// TwinCAT 3 PLC project protobuf
// Title: protobuf
// Company: TcHaxx
// Author: densogiaichned
// ProjectVersion: 0.0.0.0
// Description: Protocol Buffers for TwinCAT 3
// ProgramVersion: 3.1.4026.20
// libraries:
//   Tc2_Standard, * (Beckhoff Automation GmbH)
//   Tc2_System, * (Beckhoff Automation GmbH)
//   Tc2_Utilities, * (Beckhoff Automation GmbH)
//   TcUnit, * (www.tcunit.org)
// project tree:
//   DUTs/ E_CodedInputStreamErrorCode.TcDUT (not stored), E_CodedOutputStreamErrorCode.TcDUT (not stored), ST_ParseContext.TcDUT (not stored), ST_WriteContext.TcDUT (not stored), ST_Span.TcDUT (not stored), T_ProtobufMaxString.TcDUT (not stored), T_ProtobufRawBuffer.TcDUT (not stored)
//   FieldCodec/ FB_FieldCodec.TcPOU (not stored), FB_FieldCodecFixed32.TcPOU (not stored), FB_FieldCodecFixed64.TcPOU (not stored), FB_FieldCodecDouble.TcPOU (not stored), FB_FieldCodecBool.TcPOU (not stored), FB_FieldCodecEnum.TcPOU, FB_FieldCodecMessage.TcPOU, FB_FieldCodecUInt64.TcPOU (not stored), FB_FieldCodecUInt32.TcPOU (not stored), FB_FieldCodecString.TcPOU (not stored), FB_FieldCodecFloat.TcPOU (not stored), FB_FieldCodecInt32.TcPOU (not stored), FB_FieldCodecSint32.TcPOU (not stored), FB_FieldCodecInt64.TcPOU (not stored), FB_FieldCodecSint64.TcPOU (not stored), FB_FieldCodecBytes.TcPOU (not stored)
//   GVLs/ GCL_PB.TcGVL (not stored), Param_PB.TcGVL (not stored)
//   Helper/DUTs/ ST_VariableLengthArrayInfo.TcDUT (not stored), T_AnyInt.TcDUT (not stored), T_AnyIntOrBit.TcDUT (not stored), T_AnyString.TcDUT (not stored), T_AnyNum.TcDUT (not stored), T_Any.TcDUT (not stored), T_AnyBit.TcDUT (not stored), T_AnyBytes.TcDUT (not stored)
//   Helper/POUs/ F_ParseError.TcPOU (not stored), F_WriteError.TcPOU (not stored), F_ToAnyBit.TcPOU (not stored), F_ToAnyInt.TcPOU (not stored), F_ToAnyBytes.TcPOU (not stored), F_ToAnyType.TcPOU (not stored), F_ToAnyNum.TcPOU (not stored), F_ToAnyString.TcPOU (not stored), F_BufferInfo.TcPOU (not stored), F_WriteToBuffer.TcPOU (not stored), F_ReadFromBuffer.TcPOU (not stored)
//   ITFs/ I_Message.TcIO (not stored), I_FieldCodec.TcIO (not stored), I_RepeatedField.TcIO (not stored), I_ValueReader.TcIO (not stored), I_ValueWriter.TcIO (not stored)
//   ParsingPrimitivesMessages/POUs/ F_ReadMessage.TcPOU, F_ReadRawMessage.TcPOU (not stored), F_SkipLastField.TcPOU (not stored), F_CheckReadEndOfStreamTag.TcPOU (not stored)
//   ParsingPrimitives/DUTs/ E_ParserErrorCode.TcDUT (not stored), ST_ParserInternalState.TcDUT (not stored)
//   ParsingPrimitives/POUs/ F_DecodeZigZag32.TcPOU (not stored), F_DecodeZigZag64.TcPOU (not stored), F_MaybeConsumeTag.TcPOU (not stored), F_ParseDouble.TcPOU (not stored), F_ParseFloat.TcPOU (not stored), F_ParseRawLittleEndian32.TcPOU (not stored), F_ParseLength.TcPOU (not stored), F_ParseRawLittleEndian64.TcPOU (not stored), F_ParseRawVarint64.TcPOU (not stored), F_ParseTag.TcPOU (not stored), F_ParseRawVarint32.TcPOU (not stored), F_PeekTag.TcPOU (not stored), F_ReadBytes.TcPOU (not stored), F_ReadRawByte.TcPOU (not stored), F_ReadRawBytes.TcPOU (not stored), F_ReadStringInternal.TcPOU (not stored), F_SkipRawBytes.TcPOU (not stored), F_ReadRawString.TcPOU (not stored), F_ReadString.TcPOU (not stored)
//   / PlcTask.TcTTO (not stored), PlcTaskUnitTests.TcTTO (not stored)
//   POUs/ComputeSize/ F_ComputeBoolSize.TcPOU (not stored), F_ComputeMessageSize.TcPOU, F_ComputeTagSize.TcPOU (not stored), F_ComputeStringSize.TcPOU (not stored), F_ComputeFixed32Size.TcPOU (not stored), F_ComputeSFixed32Size.TcPOU (not stored), F_ComputeFixed64Size.TcPOU (not stored), F_ComputeSFixed64Size.TcPOU (not stored), F_ComputeInt32Size.TcPOU (not stored), F_ComputeEnumSize.TcPOU, F_ComputeFloatSize.TcPOU (not stored), F_ComputeDoubleSize.TcPOU (not stored), F_ComputeInt64Size.TcPOU (not stored), F_ComputeLengthSize.TcPOU (not stored), F_ComputeBytesSize.TcPOU (not stored), F_ComputeRawVarint64Size.TcPOU (not stored), F_ComputeSInt64Size.TcPOU (not stored), F_ComputeUInt32Size.TcPOU (not stored), F_ComputeRawVarint32Size.TcPOU (not stored), F_ComputeSInt32Size.TcPOU (not stored), F_ComputeUInt64Size.TcPOU (not stored)
//   POUs/ FB_MessageParser.TcPOU (not stored), FB_MessageWriter.TcPOU
//   POUs/ParseContext/ FB_ParseContext.TcPOU
//   POUs/SegmentedBufferHelper/ F_SbhIsReachedLimit.TcPOU (not stored), F_SbhPushLimit.TcPOU (not stored), F_SbhPopLimit.TcPOU (not stored), F_SbhRecomputeBufferSizeAfterLimit.TcPOU (not stored)
//   POUs/Span/ F_SpanFromArray.TcPOU (not stored), F_SpanSlice.TcPOU (not stored)
//   POUs/WriteContext/ FB_WriteContext.TcPOU
//   Project Information/ F_GetCompany.TcPOU (not stored), F_GetTitle.TcPOU (not stored), F_GetVersion.TcPOU (not stored)
//   RepeatedField/ FB_RepeatedField.TcPOU, F_IsPackedRepeatedField.TcPOU (not stored), F_ReadRepeatedField.TcPOU, F_WriteRepeatedField.TcPOU (not stored)
//   WireFormat/DUTs/ E_WireType.TcDUT (not stored)
//   WireFormat/GCLs/ GCL_WireFormat.TcGVL (not stored)
//   WireFormat/POus/ F_GetTagFieldNumber.TcPOU (not stored), F_GetTagWireType.TcPOU (not stored), F_MakeTag.TcPOU (not stored)
//   WritingPrimitivesMessages/POUs/ F_SetMessageValue.TcPOU (not stored), F_WriteMessage.TcPOU, F_WriteRawMessage.TcPOU (not stored)
//   WritingPrimitives/DUTs/ E_WriterErrorCode.TcDUT (not stored), ST_WriterInternalState.TcDUT (not stored)
//   WritingPrimitives/POUs/ F_EncodeZigZag32.TcPOU (not stored), F_EncodeZigZag64.TcPOU (not stored), F_WriteBytes.TcPOU (not stored), F_WriteDouble.TcPOU (not stored), F_WriteFixed32.TcPOU (not stored), F_WriteRawByte.TcPOU (not stored), F_WriteSInt32.TcPOU (not stored), F_WriteSFixed32.TcPOU (not stored), F_WriteFloat.TcPOU (not stored), F_WriteInt32.TcPOU (not stored), F_WriteFixed64.TcPOU (not stored), F_WriteSFixed64.TcPOU (not stored), F_WriteSInt64.TcPOU (not stored), F_WriteRawString.TcPOU (not stored), F_WriteRawTag.TcPOU (not stored), F_WriteUInt32.TcPOU (not stored), F_WriteRawLittleEndian32.TcPOU (not stored), F_WriteLength.TcPOU (not stored), F_WriteRawBytes.TcPOU (not stored), F_WriteRawLittleEndian64.TcPOU (not stored), F_WriteRawVarint32.TcPOU (not stored), F_WriteRawVarint64.TcPOU (not stored), F_WriteString.TcPOU (not stored), F_WriteTag.TcPOU (not stored), F_WriteEnum.TcPOU (not stored), F_WriteUInt64.TcPOU (not stored), F_WriteInt64.TcPOU (not stored)
//   __TESTs/HelperTests/ FB_F_ToAnyBytesTests.TcPOU (not stored), PRG_HelperTests.TcPOU (not stored)
//   __TESTs/EnumTests/ FB_ComputeEnumSizeTests.TcPOU, FB_FieldCodecEnumTests.TcPOU, FB_ReadEnumTests.TcPOU, FB_WriteEnumTests.TcPOU, PRG_EnumTests.TcPOU
//   __TESTs/MessagesTests/DUTs/ ST_Bar.TcDUT (not stored), ST_Baz.TcDUT (not stored), ST_Foo.TcDUT (not stored), ST_Example.TcDUT (not stored)
//   __TESTs/MessagesTests/ FB_MessageTests.TcPOU (not stored), PRG_MessageTests.TcPOU
//   __TESTs/MessagesTests/POUs/ FB_ExampleMessage.TcPOU (not stored), FB_RepeatedStringMessageTests.TcPOU (not stored), FB_RoundTripMessageExampleTest.TcPOU (not stored), FB_ReadMessageErrorTests.TcPOU, FB_TestWrongSizeMessage.TcPOU, FB_WriteMessageSizeTests.TcPOU
//   __TESTs/MessagesTests/POUs/FooBarBaz/ FB_BarMessage.TcPOU (not stored), FB_BazMessage.TcPOU (not stored), FB_FooMessage.TcPOU (not stored)
//   __TESTs/ParsingPrimitivesTests/ FB_DecodeZigZag32Tests.TcPOU (not stored), FB_DecodeZigZag64Tests.TcPOU (not stored), FB_ParseDoubleTests.TcPOU (not stored), FB_ParseFloatTests.TcPOU (not stored), FB_ParseRawVarint32Tests.TcPOU (not stored), FB_ParseRawVarint64Tests.TcPOU (not stored), FB_ReadBytesTests.TcPOU (not stored), FB_ReadRawStringTests.TcPOU (not stored), FB_ReadStringTests.TcPOU (not stored), PRG_ParsingPrimitiveTests.TcPOU (not stored)
//   __TESTs/ PRG_UnitTests.TcPOU
//   Version/ Global_Version.TcGVL (not stored)
//   __TESTs/RepeatedFieldTests/ PRG_RepeatedFieldTests.TcPOU (not stored), FB_TestFixed32Message.TcPOU
//   __TESTs/RepeatedFieldTests/Read/ FB_ReadRepeatedFieldBoolTests.TcPOU (not stored), FB_ReadRepeatedFieldBytesTests.TcPOU (not stored), FB_ReadRepeatedFieldFixed32Tests.TcPOU (not stored), FB_ReadRepeatedFieldFixed64Tests.TcPOU (not stored), FB_ReadRepeatedFieldStringTests.TcPOU (not stored), FB_ReadRepeatedFieldMessageTests.TcPOU, FB_ReadRepeatedFieldUint32Tests.TcPOU (not stored), PRG_ReadRepeatedFieldTests.TcPOU
//   __TESTs/RepeatedFieldTests/RoundTrip/ FB_RoundTripRepeatedFieldUInt32Tests.TcPOU (not stored), FB_RoundTripRepeatedFieldStringTests.TcPOU (not stored), FB_RoundTripRepeatedFieldUInt64Tests.TcPOU (not stored), PRG_RoundTripRepeatedFieldTests.TcPOU (not stored)
//   __TESTs/RepeatedFieldTests/Write/ FB_WriteRepeatedFieldBoolTests.TcPOU (not stored), FB_WriteRepeatedFieldBytesTests.TcPOU (not stored), FB_WriteRepeatedFieldDoubleTests.TcPOU (not stored), FB_WriteRepeatedFieldFixed32Tests.TcPOU (not stored), FB_WriteRepeatedFieldFixed64Tests.TcPOU (not stored), FB_WriteRepeatedFieldFloatTests.TcPOU (not stored), FB_WriteRepeatedFieldInt32Tests.TcPOU (not stored), FB_WriteRepeatedFieldInt64Tests.TcPOU (not stored), FB_WriteRepeatedFieldMessageTests.TcPOU, FB_WriteRepeatedFieldSInt32Tests.TcPOU (not stored), FB_WriteRepeatedFieldSInt64Tests.TcPOU (not stored), FB_WriteRepeatedFieldStringTests.TcPOU (not stored), FB_WriteRepeatedFieldUint32Tests.TcPOU (not stored), FB_WriteRepeatedFieldUint64Tests.TcPOU (not stored), PRG_WriteRepeatedFieldTests.TcPOU (not stored)
//   __TESTs/RoundTripTests/ FB_RoundTripBytesTests.TcPOU (not stored), FB_RoundTripFloatTests.TcPOU (not stored), FB_RoundTripDoubleTests.TcPOU (not stored), FB_RoundTripRawVarint32Tests.TcPOU (not stored), FB_RoundTripRawVarint64Tests.TcPOU (not stored), FB_RoundTripStringTests.TcPOU (not stored), FB_RoundTripTagTests.TcPOU (not stored), FB_RoundTripZigZag32Tests.TcPOU (not stored), FB_RoundTripZigZag64Tests.TcPOU (not stored), PRG_RoundTripTests.TcPOU (not stored)
//   __TESTs/SpanTests/ FB_F_SpanFromArrayTests.TcPOU (not stored), FB_F_SpanSliceTests.TcPOU (not stored), PRG_SpanTests.TcPOU (not stored)
//   __TESTs/WireFormatTests/ FB_MakeTagTests.TcPOU (not stored), PRG_WireFormatTests.TcPOU (not stored)
//   __TESTs/WritingPrimitiveTests/ FB_EncodeZigZag64Tests.TcPOU (not stored), FB_EncodeZigZag32Tests.TcPOU (not stored), FB_WriteBytesTests.TcPOU (not stored), FB_WriteDoubleTests.TcPOU (not stored), FB_WriteRawVarint32Tests.TcPOU (not stored), FB_WriteFloatTests.TcPOU (not stored), FB_WriteRawVarint64Tests.TcPOU (not stored), FB_WriteTagTests.TcPOU (not stored), FB_WriteStringTests.TcPOU (not stored), PRG_WritingPrimitiveTests.TcPOU (not stored)
//   __TESTs/__GENERATED/ E_Color.TcDUT (not stored), E_DataType.TcDUT (not stored), E_Status.TcDUT (not stored), FB_ComplexData.TcPOU (not stored), FB_Device.TcPOU (not stored), FB_Motor.TcPOU (not stored), FB_MotorConfig.TcPOU (not stored), FB_ScalarTypesTest.TcPOU (not stored), FB_SensorReading.TcPOU (not stored), ST_ComplexData.TcDUT (not stored), ST_Device.TcDUT (not stored), ST_Motor.TcDUT (not stored), ST_MotorConfig.TcDUT (not stored), ST_ScalarTypesTest.TcDUT (not stored), ST_SensorReading.TcDUT (not stored)

// ---- FieldCodec/FB_FieldCodecEnum.TcPOU
FUNCTION_BLOCK FB_FieldCodecEnum EXTENDS FB_FieldCodec
VAR_INPUT
END_VAR
VAR_OUTPUT
END_VAR
VAR
    nValue : DINT;
END_VAR

METHOD CalculatePackedDataSize : HRESULT
VAR_INPUT CONSTANT
	anyFirstElem	: T_Any;
	nLength	        : UDINT;
END_VAR
VAR_OUTPUT
    nPackedDataSize : UDINT;
END_VAR
VAR
    anyItem : T_Any;
    i : UDINT;
    nCopySize : UDINT;
    nTmp : DINT;
    retVal : UDINT;
END_VAR
nPackedDataSize := 0;

IF anyFirstElem.pValue = NULL OR anyFirstElem.TypeClass <> __SYSTEM.TYPE_CLASS.TYPE_ENUM THEN
    CalculatePackedDataSize := E_HRESULTAdsErr.INVALIDDATA;
    RETURN;
END_IF

nCopySize := MIN(TO_UDINT(anyFirstElem.diSize), SIZEOF(nTmp));
IF nCopySize = 0 THEN
    CalculatePackedDataSize := E_HRESULTAdsErr.INVALIDDATA;
    RETURN;
END_IF

IF nLength < 1 THEN
    CalculatePackedDataSize := S_OK;
    RETURN;
END_IF

anyItem := anyFirstElem;

FOR i := 0 TO nLength - 1 DO
    anyItem.pValue := anyFirstElem.pValue + (i * TO_UDINT(anyFirstElem.diSize));
    nTmp := 0;
    retVal := MEMCPY(destAddr:= ADR(nTmp), srcAddr:= anyItem.pValue, n:= nCopySize);
    IF retVal = 0 THEN
        CalculatePackedDataSize := E_HRESULTAdsErr.INVALIDDATA;
        RETURN;
    END_IF
    nPackedDataSize := nPackedDataSize + F_ComputeInt32Size(nTmp);
END_FOR

CalculatePackedDataSize := S_OK;
END_METHOD

METHOD IsPackedRepeatedField : BOOL
VAR_INPUT
	nTag	: UDINT;
END_VAR
IsPackedRepeatedField := F_IsPackedRepeatedField(nTag);
END_METHOD


METHOD ValueReader : HRESULT
VAR_IN_OUT
    stCtx : ST_ParseContext;
END_VAR
VAR_OUTPUT
	anyOut	: T_Any;
END_VAR
nValue := 0;
ValueReader := F_ParseRawVarint32(stCtx, nValue);
IF FAILED(ValueReader) THEN
    RETURN;
END_IF

anyOut := F_ToAnyType(anyArg:= nValue);
END_METHOD

METHOD ValueWriter : HRESULT
VAR_IN_OUT
    stCtx  : ST_WriteContext;
END_VAR
VAR_INPUT
	anyIn	: T_ANY;
END_VAR
VAR
    nCopySize : UDINT;
    retVal : UDINT;
END_VAR
IF anyIn.pValue = NULL OR anyIn.TypeClass <> __SYSTEM.TYPE_CLASS.TYPE_ENUM THEN
    ValueWriter := E_HRESULTAdsErr.INVALIDDATA;
    RETURN;
END_IF

nCopySize := MIN(TO_UDINT(anyIn.diSize), SIZEOF(nValue));
IF nCopySize = 0 THEN
    ValueWriter := E_HRESULTAdsErr.INVALIDDATA;
    RETURN;
END_IF

nValue := 0;
retVal := MEMCPY(destAddr:= ADR(nValue), srcAddr:= anyIn.pValue, n:= nCopySize);
IF retVal = 0 THEN
    ValueWriter := E_HRESULTAdsErr.INVALIDDATA;
    RETURN;
END_IF

ValueWriter := F_WriteEnum(stCtx, nValue);
END_METHOD

END_FUNCTION_BLOCK

// ---- FieldCodec/FB_FieldCodecMessage.TcPOU
FUNCTION_BLOCK FB_FieldCodecMessage Extends FB_FieldCodec
VAR_INPUT
END_VAR
VAR_OUTPUT
END_VAR
VAR
END_VAR

{attribute 'analysis' := '-33'}
METHOD CalculatePackedDataSize : HRESULT
VAR_INPUT CONSTANT
	anyFirstElem	: T_Any;
	nLength	        : UDINT;        // items to write
END_VAR
VAR_OUTPUT
    nPackedDataSize : UDINT;
END_VAR
VAR
    anyItem : T_Any;
    i : UDINT;
    eErrorCode : E_WriterErrorCode;
END_VAR
nPackedDataSize := 0;

IF THIS^.ipMessageField = NULL THEN
    CalculatePackedDataSize := E_HRESULTAdsErr.INVALIDDATA;
    RETURN;
END_IF

IF nLength < 1 THEN
    CalculatePackedDataSize := S_OK;
    RETURN;
END_IF

anyItem := anyFirstElem;

FOR i := 0 TO nLength - 1 DO
    anyItem.pValue := anyFirstElem.pValue + (i * TO_UDINT(anyFirstElem.diSize));
    eErrorCode := F_SetMessageValue(anyValue:= anyItem, iMessage:= THIS^.ipMessageField);
    IF FAILED(eErrorCode) THEN
        CalculatePackedDataSize := E_HRESULTAdsErr.INVALIDDATA;
        RETURN;
    END_IF

    nPackedDataSize := nPackedDataSize + F_ComputeMessageSize(iMessage:= THIS^.ipMessageField);
END_FOR

CalculatePackedDataSize := S_OK;
END_METHOD

//FB_Init is always available implicitly and it is used primarily for initialization.
//The return value is not evaluated. For a specific influence, you can also declare the
//methods explicitly and provide additional code there with the standard initialization
//code. You can evaluate the return value.
METHOD FB_Init: BOOL
VAR_INPUT
    bInitRetains: BOOL; // TRUE: the retain variables are initialized (reset warm / reset cold)
    bInCopyCode: BOOL;  // TRUE: the instance will be copied to the copy code afterward (online change)
	nTag : UDINT;	
	ipMessage : I_Message;
END_VAR
nTagField := nTag;
ipMessageField := ipMessage;
END_METHOD

METHOD IsPackedRepeatedField : BOOL
VAR_INPUT
    {attribute 'analysis' := '-33' } 
	nTag	: UDINT;
END_VAR

IsPackedRepeatedField := FALSE;
END_METHOD


METHOD ValueReader : HRESULT
VAR_IN_OUT      
    stCtx : ST_ParseContext;
END_VAR
VAR_OUTPUT
	anyOut	: T_Any;
END_VAR

IF stCtx.pCurrentContext = NULL THEN
    ValueReader := F_ParseError(stCtx, E_ParserErrorCode.InternalError);
    RETURN;
END_IF

stCtx.pCurrentContext^.InitializeFromState(stBuffer:= stCtx.stBuffer, stState:= stCtx.stState);
ValueReader := F_ReadMessage(fbCtx:= stCtx.pCurrentContext^, iMessage:= THIS^.ipMessageField);
anyOut := THIS^.ipMessageField.MessageValue;
stCtx.stState := stCtx.pCurrentContext^.refCtx.stState;
END_METHOD

METHOD ValueWriter : HRESULT
VAR_IN_OUT
    stCtx  : ST_WriteContext;
END_VAR
VAR_INPUT
    anyIn : T_ANY;
END_VAR
VAR
	eErrorCode : E_WriterErrorCode;
END_VAR

// IF THIS^.pWriteContextField = NULL THEN
//     ValueWriter := F_WriteError(stCtx, E_WriterErrorCode.InternalError);
//     RETURN;
// END_IF
// 
// THIS^.pWriteContextField^.InitializeFromState(stBuffer:= stCtx.stBuffer, stState:= stCtx.stState);


eErrorCode := F_SetMessageValue(anyValue:= anyIn, iMessage:= THIS^.ipMessageField);
IF FAILED(eErrorCode) THEN
	F_WriteError(stCtx, eErrorCode);
	RETURN;
END_IF

// ValueWriter := F_WriteMessage(fbCtx:= THIS^.pWriteContextField^, THIS^.ipMessageField);
ValueWriter := F_WriteMessage(stCtx:= stCtx, THIS^.ipMessageField);
END_METHOD

END_FUNCTION_BLOCK

// ---- POUs/ComputeSize/F_ComputeMessageSize.TcPOU
{attribute 'estimated-stack-usage' := '8192'}
// Computes the number of bytes that would be needed to encode an
// embedded message field, including the tag.
FUNCTION F_ComputeMessageSize : UDINT
VAR_INPUT
    iMessage : I_Message;
END_VAR
VAR
	nSize	: UDINT;
    aBuffer : T_ProtobufRawBuffer;
    hr : HRESULT;
END_VAR


IF iMessage = NULL THEN
	RETURN;
END_IF

hr := iMessage.Writer.WriteTo(aBuffer);
IF FAILED(hr) THEN
    RETURN;
END_IF

nSize := iMessage.Writer.nBytesWritten;
F_ComputeMessageSize := F_ComputeLengthSize(nSize) + nSize;

END_FUNCTION

// ---- ParsingPrimitivesMessages/POUs/F_ReadMessage.TcPOU
FUNCTION F_ReadMessage : HRESULT
VAR_IN_OUT
    fbCtx   : FB_ParseContext;     
END_VAR
VAR_INPUT
    iMessage : I_Message;
END_VAR
VAR
    nLength, nOldLength : UDINT;
END_VAR


F_ReadMessage := F_ParseLength(fbCtx.refCtx, nLength=> nLength);
IF FAILED(F_ReadMessage) THEN
    RETURN;
END_IF

IF fbCtx.refCtx.stState.nRecursionDepth >= fbCtx.refCtx.stState.nRecursionLimit THEN
    F_ReadMessage := fbCtx.refCtx.stState.eParserErrorCode := E_ParserErrorCode.RecursionLimitExceeded;
    fbCtx.refCtx.stState.bError := TRUE;
    RETURN;
END_IF


F_ReadMessage := F_SbhPushLimit(fbCtx.refCtx.stState, nLength, nCurrentLimit=> nOldLength);
IF FAILED(F_ReadMessage) THEN
    RETURN;
END_IF

fbCtx.refCtx.stState.nRecursionDepth := fbCtx.refCtx.stState.nRecursionDepth + 1;
F_ReadMessage := F_ReadRawMessage(fbCtx, iMessage);
IF FAILED(F_ReadMessage) THEN
    RETURN;
END_IF

F_ReadMessage := F_CheckReadEndOfStreamTag(fbCtx.refCtx.stState);
IF FAILED(F_ReadMessage) THEN
    RETURN;
END_IF

IF NOT F_SbhIsReachedLimit(fbCtx.refCtx.stState) THEN
    F_ReadMessage := fbCtx.refCtx.stState.eParserErrorCode := E_ParserErrorCode.TruncatedMessage;
    fbCtx.refCtx.stState.bError := TRUE;
    RETURN;
END_IF

fbCtx.refCtx.stState.nRecursionDepth := fbCtx.refCtx.stState.nRecursionDepth - 1;
F_ReadMessage := F_SbhPopLimit(fbCtx.refCtx.stState, nOldLength);

END_FUNCTION

// ---- POUs/ParseContext/FB_ParseContext.TcPOU
// Represents the current parsing state and is passed along
// as the parsing proceeds.
// All the public methods are intended to be invoked only by the generated code,
// users should never invoke them directly.
{attribute 'no_explicit_call' := 'do not call this POU directly'} 
FUNCTION_BLOCK FINAL FB_ParseContext
VAR_INPUT
END_VAR
VAR_OUTPUT
END_VAR
VAR
    stCtx   : ST_ParseContext;
END_VAR

VAR
END_VAR

// Internal-only property; when set to true, unknown fields will be discarded while parsing.
PROPERTY INTERNAL DiscardUnknownFields : BOOL
GET
DiscardUnknownFields := stCtx.stState.bDiscardUnknownFields;
END_GET
SET
stCtx.stState.bDiscardUnknownFields := DiscardUnknownFields;
END_SET
END_PROPERTY

METHOD FromBuffer : HRESULT
VAR_IN_OUT CONSTANT
    aBuffer : ARRAY [*] OF BYTE;
END_VAR

Reset();
Initialize(F_SpanFromArray(aBuffer));
END_METHOD

METHOD INTERNAL Initialize
VAR_INPUT CONSTANT
    stBuffer    : ST_Span;    
END_VAR
stCtx.stBuffer := stBuffer;

stCtx.stState.nBufferSize       := stBuffer.nSize;
stCtx.stState.nSizeLimit        := Param_PB.cMaxProtobufRawBuffer;
stCtx.stState.nRecursionLimit   := Param_PB.cRecursionLimit; 
stCtx.stState.nCurrentLimit     := TO_UDINT(-1);

stCtx.pCurrentContext 			:= THIS;
END_METHOD

// Initialize a ST_ParseContext using existing ST_ParserInternalState,
METHOD INTERNAL InitializeFromState
VAR_IN_OUT CONSTANT
    stState : ST_ParserInternalState;
    stBuffer : ST_Span;    
END_VAR
THIS^.stCtx.stState  := stState;
THIS^.stCtx.stBuffer := stBuffer;

stCtx.pCurrentContext := THIS;
END_METHOD

// Returns the last tag read, OR 0 IF no tags have been read OR we've read beyond the end of the input.
PROPERTY INTERNAL LastTag : UDINT
GET
LastTag := stCtx.stState.nLastTag;
END_GET
END_PROPERTY

METHOD ReadBool : HRESULT
VAR_OUTPUT
    bValue : BOOL;
END_VAR
VAR
    nTmp : BYTE;
END_VAR

ReadBool := F_ParseRawVarint32(THIS^.stCtx, nTmp);
bValue := nTmp <> 0;
END_METHOD

METHOD ReadBytes : HRESULT
VAR_IN_OUT
    aBytes : ARRAY [*] OF BYTE;
END_VAR
VAR_OUTPUT
	nCount : UDINT;
END_VAR

ReadBytes := F_ReadBytes(THIS^.stCtx, aBytes, nLength=> nCount);
END_METHOD

METHOD PUBLIC ReadDouble : HRESULT
VAR_OUTPUT
    fValue : LREAL;
END_VAR

ReadDouble := F_ParseDouble(THIS^.stCtx, fValue=> fValue);
END_METHOD

METHOD PUBLIC ReadEnum : HRESULT
VAR_INPUT
    anyEnum : ANY;
END_VAR
VAR
    nTmp   : UDINT;
	nCopySize : UDINT;
	retVal : UDINT;
END_VAR
IF anyEnum.pValue = NULL OR anyEnum.TypeClass <> __SYSTEM.TYPE_CLASS.TYPE_ENUM THEN
	ReadEnum := E_HRESULTAdsErr.INVALIDDATA;
	RETURN;
END_IF

ReadEnum := F_ParseRawVarint32(THIS^.stCtx, nTmp);
IF FAILED(ReadEnum) THEN
	RETURN;
END_IF

nCopySize := MIN(TO_UDINT(anyEnum.diSize), SIZEOF(nTmp));
IF nCopySize = 0 THEN
	ReadEnum := E_HRESULTAdsErr.INVALIDDATA;
	RETURN;
END_IF

MEMSET(destAddr:= anyEnum.pValue, fillByte:= 16#0, n:= TO_UDINT(anyEnum.diSize));
retVal := MEMCPY(destAddr:= anyEnum.pValue, srcAddr:= ADR(nTmp), n:= nCopySize);
IF retVal = 0 THEN
	ReadEnum := E_HRESULTAdsErr.INVALIDDATA;
END_IF
END_METHOD

METHOD PUBLIC ReadFixed32 : HRESULT
VAR_OUTPUT
    nValue : UDINT;
END_VAR

ReadFixed32 := F_ParseRawLittleEndian32(THIS^.stCtx, nValue=> nValue);
END_METHOD

METHOD PUBLIC ReadFixed64 : HRESULT
VAR_OUTPUT
    nValue : ULINT;
END_VAR

ReadFixed64 := F_ParseRawLittleEndian64(THIS^.stCtx, nValue=> nValue);
END_METHOD

METHOD PUBLIC ReadFloat : HRESULT
VAR_OUTPUT
    fValue : REAL;
END_VAR

ReadFloat := F_ParseFloat(THIS^.stCtx, fValue=> fValue);
END_METHOD

METHOD PUBLIC ReadInt32 : HRESULT
VAR_INPUT
    anyDint : ANY;
END_VAR
VAR
    nTmp   : UDINT;
	retVal : UDINT;
END_VAR

ReadInt32 := F_ParseRawVarint32(THIS^.stCtx, nTmp);
retVal := memcpy(destAddr:= anyDint.pValue, srcAddr:= ADR(nTmp), n:= MIN(TO_UDINT(anyDint.diSize), SIZEOF(nTmp)));
IF retVal = 0 THEN
	ReadInt32:= E_HRESULTAdsErr.INVALIDDATA;
END_IF
END_METHOD

METHOD PUBLIC ReadInt64 : HRESULT
VAR_INPUT
    anyLint : ANY;
END_VAR
VAR
    nTmp   : ULINT;
	retVal : UDINT;
END_VAR

ReadInt64 := F_ParseRawVarint64(THIS^.stCtx, nTmp);
retVal := memcpy(destAddr:= anyLint.pValue, srcAddr:= ADR(nTmp), n:= MIN(TO_UDINT(anyLint.diSize), SIZEOF(nTmp)));
IF retVal = 0 THEN
	ReadInt64:= E_HRESULTAdsErr.INVALIDDATA;
END_IF
END_METHOD

// Reads a length for length-delimited data.
METHOD PUBLIC ReadLength : HRESULT
VAR_OUTPUT
    nLength : UDINT;
END_VAR
ReadLength := F_ParseLength(THIS^.stCtx, nLength=> nLength);
END_METHOD

METHOD ReadMessage : HRESULT
VAR_INPUT
    ipMessage : I_Message;
END_VAR

ReadMessage := F_ReadMessage(fbCtx:= THIS^, ipMessage);
END_METHOD

METHOD PUBLIC ReadSFixed32 : HRESULT
VAR_OUTPUT
    nValue : DINT;
END_VAR
VAR
    nTmp : UDINT;
END_VAR

ReadSFixed32 := F_ParseRawLittleEndian32(THIS^.stCtx, nValue=> nTmp);

nValue := TO_DINT(nTmp);
END_METHOD

METHOD PUBLIC ReadSFixed64 : HRESULT
VAR_OUTPUT
    nValue : LINT;
END_VAR
VAR
    nTmp : ULINT;
END_VAR

ReadSFixed64 := F_ParseRawLittleEndian64(THIS^.stCtx, nValue=> nTmp);

nValue := TO_LINT(nTmp);
END_METHOD

METHOD PUBLIC ReadSInt32 : HRESULT
VAR_INPUT
    anyDint : ANY;
END_VAR
VAR
    nTmp   : UDINT;
	nValue : DINT;
	retVal : UDINT;
END_VAR

ReadSInt32 := F_ParseRawVarint32(THIS^.stCtx, nTmp);
nValue := F_DecodeZigZag32(nTmp);
retVal := memcpy(destAddr:= anyDint.pValue, srcAddr:= ADR(nValue), n:= MIN(TO_UDINT(anyDint.diSize), SIZEOF(nValue)));
IF retVal = 0 THEN
	ReadSInt32:= E_HRESULTAdsErr.INVALIDDATA;
END_IF
END_METHOD

METHOD PUBLIC ReadSInt64 : HRESULT
VAR_INPUT
    anyLint : ANY;
END_VAR
VAR
    nTmp   : ULINT;
	nValue : LINT;
	retVal : UDINT;
END_VAR

ReadSInt64 := F_ParseRawVarint64(THIS^.stCtx, nTmp);
nValue := F_DecodeZigZag64(nTmp);
retVal := memcpy(destAddr:= anyLint.pValue, srcAddr:= ADR(nValue), n:= MIN(TO_UDINT(anyLint.diSize), SIZEOF(nValue)));
IF retVal = 0 THEN
	ReadSInt64:= E_HRESULTAdsErr.INVALIDDATA;
END_IF
END_METHOD

METHOD PUBLIC ReadString : HRESULT
VAR_INPUT
    anyStringOut : ANY_STRING;
END_VAR
ReadString := F_ReadString(THIS^.stCtx, F_ToAnyType(anyStringOut));
END_METHOD

// Peeks at the next field tag. this is like calling "ReadTag", but the
// tag is not consumed. (So a subsequent call to "ReadTag" will return the same value.)
METHOD PUBLIC ReadTag : HRESULT
VAR_OUTPUT
    nTag : UDINT;
END_VAR
ReadTag := F_ParseTag(THIS^.stCtx, nTag=>nTag);
END_METHOD

METHOD PUBLIC ReadUint32 : HRESULT
VAR_INPUT
    anyUdint : ANY;
END_VAR
VAR
    nTmp   : UDINT;
	retVal : UDINT;
END_VAR

ReadUint32 := F_ParseRawVarint32(THIS^.stCtx, nTmp);
retVal := memcpy(destAddr:= anyUdint.pValue, srcAddr:= ADR(nTmp), n:= MIN(TO_UDINT(anyUdint.diSize), SIZEOF(nTmp)));
IF retVal = 0 THEN
	ReadUint32:= E_HRESULTAdsErr.INVALIDDATA;
END_IF
END_METHOD

METHOD PUBLIC ReadUint64 : HRESULT
VAR_INPUT
    anyUlint : ANY;
END_VAR
VAR
    nTmp   : ULINT;
	retVal : UDINT;
END_VAR

ReadUint64 := F_ParseRawVarint64(THIS^.stCtx, nTmp);
retVal := memcpy(destAddr:= anyUlint.pValue, srcAddr:= ADR(nTmp), n:= MIN(TO_UDINT(anyUlint.diSize), SIZEOF(nTmp)));
IF retVal = 0 THEN
	ReadUint64:= E_HRESULTAdsErr.INVALIDDATA;
END_IF
END_METHOD

PROPERTY refCtx : REFERENCE TO ST_ParseContext
GET
refCtx REF= THIS^.stCtx ;
END_GET
END_PROPERTY

METHOD PRIVATE Reset
VAR_INPUT
END_VAR

stCtx.stState.bError := FALSE;
stCtx.stState.eParserErrorCode := S_OK;
stCtx.stState.nBufferPos := 0;
stCtx.stState.nBufferSize := 0;
END_METHOD

METHOD SkipLastField : HRESULT
VAR_INPUT
END_VAR

SkipLastField := F_SkipLastField(THIS^.stCtx);
END_METHOD

END_FUNCTION_BLOCK

// ---- WritingPrimitivesMessages/POUs/F_WriteMessage.TcPOU
{attribute 'estimated-stack-usage' := '8192'}
// Writes a message, without a tag. The data is length-prefixed.
FUNCTION F_WriteMessage : HRESULT
VAR_IN_OUT
//     fbCtx   : FB_WriteContext;
	stCtx : ST_WriteContext;     
END_VAR
VAR_INPUT
    ipMessage : I_Message;
END_VAR
VAR
    nLength : UDINT;
    aPayload : T_ProtobufRawBuffer;
END_VAR

IF ipMessage = NULL THEN
	F_WriteMessage := F_WriteError(stCtx:= stCtx, eError:= E_WriterErrorCode.InternalError);
	RETURN;
END_IF

F_WriteMessage := ipMessage.Writer.WriteTo(aPayload);
IF FAILED(F_WriteMessage) THEN
	RETURN;
END_IF

nLength := ipMessage.Writer.nBytesWritten;
F_WriteMessage := F_WriteLength(stCtx:= stCtx, nLength:= nLength);
IF FAILED(F_WriteMessage) THEN
	RETURN;
END_IF

F_WriteMessage := F_WriteRawBytes(stCtx:= stCtx, tBytes:= F_ToAnyBytes(aPayload), nLength:= nLength);

END_FUNCTION

// ---- POUs/ComputeSize/F_ComputeEnumSize.TcPOU
FUNCTION F_ComputeEnumSize : UDINT
VAR_INPUT
    anyEnum  : ANY;
END_VAR
VAR
	nTmp : DINT;
	nCopySize : UDINT;
END_VAR

IF anyEnum.pValue = NULL OR anyEnum.TypeClass <> __SYSTEM.TYPE_CLASS.TYPE_ENUM THEN
	RETURN;
END_IF

nCopySize := MIN(TO_UDINT(anyEnum.diSize), SIZEOF(nTmp));
IF nCopySize = 0 THEN
	RETURN;
END_IF

nTmp := 0;
MEMCPY(destAddr:= ADR(nTmp), srcAddr:= anyEnum.pValue, n:= nCopySize);
F_ComputeEnumSize := F_ComputeInt32Size(nTmp);

END_FUNCTION

// ---- POUs/FB_MessageWriter.TcPOU
FUNCTION_BLOCK PUBLIC FINAL FB_MessageWriter
VAR_INPUT
END_VAR
VAR_OUTPUT
END_VAR
VAR
    fbWriteCtx  : FB_WriteContext;
    ipMessage   : I_Message;
    nBytesWrittenField : UDINT;
END_VAR

//FB_Init is always available implicitly and it is used primarily for initialization.
//The return value is not evaluated. For a specific influence, you can also declare the
//methods explicitly and provide additional code there with the standard initialization
//code. You can evaluate the return value.
METHOD FB_Init: BOOL
VAR_INPUT
    bInitRetains: BOOL; // TRUE: the retain variables are initialized (reset warm / reset cold)
    bInCopyCode: BOOL;  // TRUE: the instance will be copied to the copy code afterward (online change)
    ipMessage   : I_Message;
END_VAR
THIS^.ipMessage := ipMessage;
END_METHOD

PROPERTY nBytesWritten : UDINT
GET
nBytesWritten := THIS^.nBytesWrittenField;
END_GET
END_PROPERTY

METHOD PUBLIC WriteTo : HRESULT
VAR_IN_OUT CONSTANT
    aBuffer     : ARRAY[*] OF BYTE;
END_VAR

nBytesWrittenField := 0;

IF ipMessage = 0 THEN
    WriteTo := E_WriterErrorCode.InternalError;
    RETURN;
END_IF

WriteTo := fbWriteCtx.FromBuffer(aBuffer);
IF FAILED(WriteTo) THEN
    RETURN;
END_IF

WriteTo := ipMessage.WriteTo(fbWriteCtx:= fbWriteCtx);
IF SUCCEEDED(WriteTo) THEN
    nBytesWrittenField := fbWriteCtx.refCtx.stState.nBufferPos;
END_IF
END_METHOD

END_FUNCTION_BLOCK

// ---- POUs/WriteContext/FB_WriteContext.TcPOU
// Represents the current serialization state and is passed along
// as the serialization proceeds.
// All the public methods are intended to be invoked only by the generated code,
// users should never invoke them directly.
{attribute 'no_explicit_call' := 'do not call this POU directly'} 
FUNCTION_BLOCK PUBLIC FINAL FB_WriteContext
VAR
    stCtx   : ST_WriteContext;
END_VAR

VAR
END_VAR

METHOD FromBuffer : HRESULT
VAR_IN_OUT CONSTANT
    aBuffer : ARRAY [*] OF BYTE;
END_VAR

Reset();
Initialize(F_SpanFromArray(aBuffer));
END_METHOD

METHOD INTERNAL Initialize
VAR_INPUT CONSTANT
    stBuffer    : ST_Span;    
END_VAR
stCtx.stBuffer := stBuffer;

stCtx.stState.nBufferSize        := stBuffer.nSize;
stCtx.stState.nBufferPos         := 0;

stCtx.pCurrentContext			:= THIS;
END_METHOD

// Initialize a ST_WriterContext using existing ST_WriterInternalState,
METHOD INTERNAL InitializeFromState
VAR_IN_OUT CONSTANT
    stBuffer : ST_Span;
    stState : ST_WriterInternalState;        
END_VAR
THIS^.stCtx.stState  := stState;
THIS^.stCtx.stBuffer := stBuffer;

stCtx.pCurrentContext := THIS;
END_METHOD

PROPERTY nSpaceLeft : UDINT
GET
nSpaceLeft := stCtx.stState.nBufferSize - stCtx.stState.nBufferPos;
END_GET
END_PROPERTY

PROPERTY refCtx : REFERENCE TO ST_WriteContext
GET
refCtx REF= THIS^.stCtx ;
END_GET
END_PROPERTY

METHOD PRIVATE Reset
VAR_INPUT
END_VAR

stCtx.stState.bError := FALSE;
stCtx.stState.eWriterErrorCode := S_OK;
stCtx.stState.nBufferPos := 0;
stCtx.stState.nBufferSize := 0;
END_METHOD

METHOD WriteBool : HRESULT
VAR_INPUT
    bValue : BOOL;
END_VAR

WriteBool := F_WriteRawByte(THIS^.stCtx, TO_BYTE(bValue));
END_METHOD

METHOD WriteBytes : HRESULT
VAR_IN_OUT CONSTANT
    aBytes  : ARRAY [*] OF BYTE;
END_VAR
VAR_INPUT
    nCount : UDINT;
END_VAR

WriteBytes := F_WriteBytes(THIS^.stCtx, aBytes, nCount);
END_METHOD

METHOD WriteDouble : HRESULT
VAR_INPUT
    fValue : LREAL;
END_VAR
WriteDouble := F_WriteDouble(THIS^.stCtx, fValue);
END_METHOD

METHOD WriteEnum : HRESULT
VAR_INPUT
    anyEnum : ANY;
END_VAR
VAR
	nTmp : DINT;
	nCopySize : UDINT;
	retVal : UDINT;
END_VAR
IF anyEnum.pValue = NULL OR anyEnum.TypeClass <> __SYSTEM.TYPE_CLASS.TYPE_ENUM THEN
	WriteEnum := E_HRESULTAdsErr.INVALIDDATA;
	RETURN;
END_IF

nCopySize := MIN(TO_UDINT(anyEnum.diSize), SIZEOF(nTmp));
IF nCopySize = 0 THEN
	WriteEnum := E_HRESULTAdsErr.INVALIDDATA;
	RETURN;
END_IF

nTmp := 0;
retVal := MEMCPY(destAddr:= ADR(nTmp), srcAddr:= anyEnum.pValue, n:= nCopySize);
IF retVal = 0 THEN
	WriteEnum := E_HRESULTAdsErr.INVALIDDATA;
	RETURN;
END_IF

WriteEnum := F_WriteEnum(THIS^.stCtx, nTmp);
END_METHOD

METHOD WriteFixed32 : HRESULT
VAR_INPUT
    nValue : UDINT;
END_VAR

WriteFixed32 := F_WriteFixed32(THIS^.stCtx, nValue);
END_METHOD

METHOD WriteFixed64 : HRESULT
VAR_INPUT
    nValue : ULINT;
END_VAR

WriteFixed64 := F_WriteFixed64(THIS^.stCtx, nValue);
END_METHOD

METHOD WriteFloat : HRESULT
VAR_INPUT
    fValue : REAL;
END_VAR
WriteFloat := F_WriteFloat(THIS^.stCtx, fValue);
END_METHOD

METHOD WriteInt32 : HRESULT
VAR_INPUT
    anyDint : ANY;
END_VAR
VAR
    nTmp   : DINT;
	retVal : UDINT;
END_VAR

retVal := memcpy(destAddr:= ADR(nTmp), srcAddr:= anyDint.pValue, n:= MIN(TO_UDINT(anyDint.diSize), SIZEOF(nTmp)));
IF retVal = 0 THEN
	WriteInt32:= E_HRESULTAdsErr.INVALIDDATA;
	RETURN;
END_IF

WriteInt32 := F_WriteInt32(THIS^.stCtx, nTmp);
END_METHOD

METHOD WriteInt64 : HRESULT
VAR_INPUT
    anyLint : ANY;
END_VAR
VAR
    nTmp   : LINT;
	retVal : UDINT;
END_VAR

retVal := memcpy(destAddr:= ADR(nTmp), srcAddr:= anyLint.pValue, n:= MIN(TO_UDINT(anyLint.diSize), SIZEOF(nTmp)));
IF retVal = 0 THEN
	WriteInt64:= E_HRESULTAdsErr.INVALIDDATA;
	RETURN;
END_IF

WriteInt64 := F_WriteInt64(THIS^.stCtx, nTmp);
END_METHOD

METHOD WriteLength : HRESULT
VAR_INPUT
    nLength : UDINT;
END_VAR

WriteLength := F_WriteLength(THIS^.stCtx, nLength);
END_METHOD

METHOD WriteMessage : HRESULT
VAR_INPUT
    ipMessage : I_Message;
END_VAR

WriteMessage := F_WriteMessage(stCtx:= THIS^.stCtx, ipMessage);
END_METHOD

METHOD WriteRawTag : HRESULT
VAR_INPUT
	nTag    : UDINT;
END_VAR
WriteRawTag := F_WriteRawTag(THIS^.stCtx, nTag);
END_METHOD

METHOD WriteSFixed32 : HRESULT
VAR_INPUT
    nValue : DINT;
END_VAR

WriteSFixed32 := F_WriteSFixed32(THIS^.stCtx, nValue);
END_METHOD

METHOD WriteSFixed64 : HRESULT
VAR_INPUT
    nValue : LINT;
END_VAR

WriteSFixed64 := F_WriteSFixed64(THIS^.stCtx, nValue);
END_METHOD

METHOD WriteSint32 : HRESULT
VAR_INPUT
    anyDint : ANY;
END_VAR
VAR
    nTmp   : DINT;
	retVal : UDINT;
END_VAR

retVal := memcpy(destAddr:= ADR(nTmp), srcAddr:= anyDint.pValue, n:= MIN(TO_UDINT(anyDint.diSize), SIZEOF(nTmp)));
IF retVal = 0 THEN
	WriteSint32:= E_HRESULTAdsErr.INVALIDDATA;
	RETURN;
END_IF

WriteSint32 := F_WriteSInt32(THIS^.stCtx, nTmp);
END_METHOD

METHOD WriteSint64 : HRESULT
VAR_INPUT
    anyLint : ANY;
END_VAR
VAR
    nTmp   : LINT;
	retVal : UDINT;
END_VAR

retVal := memcpy(destAddr:= ADR(nTmp), srcAddr:= anyLint.pValue, n:= MIN(TO_UDINT(anyLint.diSize), SIZEOF(nTmp)));
IF retVal = 0 THEN
	WriteSint64:= E_HRESULTAdsErr.INVALIDDATA;
	RETURN;
END_IF

WriteSint64 := F_WriteSInt64(THIS^.stCtx, nTmp);
END_METHOD

METHOD WriteString : HRESULT
VAR_IN_OUT CONSTANT
    sStringToWrite          : T_ProtobufMaxString;
END_VAR

WriteString := F_WriteString(THIS^.stCtx, sStringToWrite);
END_METHOD

METHOD WriteTag : HRESULT
VAR_INPUT
    nFieldNumber    : UDINT;
    eWireType       : E_WireType;
END_VAR

WriteTag := F_WriteTag(THIS^.stCtx, nFieldNumber, eWireType);
END_METHOD

METHOD WriteUint32 : HRESULT
VAR_INPUT
    anyUdint : ANY;
END_VAR
VAR
    nTmp   : UDINT;
	retVal : UDINT;
END_VAR


retVal := memcpy(destAddr:= ADR(nTmp), srcAddr:= anyUdint.pValue, n:= MIN(TO_UDINT(anyUdint.diSize), SIZEOF(nTmp)));
IF retVal = 0 THEN
	WriteUint32:= E_HRESULTAdsErr.INVALIDDATA;
	RETURN;
END_IF

WriteUint32 := F_WriteUInt32(THIS^.stCtx, nTmp);
END_METHOD

METHOD WriteUint64 : HRESULT
VAR_INPUT
    anyUlint : ANY;
END_VAR
VAR
    nTmp   : ULINT;
	retVal : UDINT;
END_VAR

retVal := memcpy(destAddr:= ADR(nTmp), srcAddr:= anyUlint.pValue, n:= MIN(TO_UDINT(anyUlint.diSize), SIZEOF(nTmp)));
IF retVal = 0 THEN
	WriteUint64:= E_HRESULTAdsErr.INVALIDDATA;
	RETURN;
END_IF

WriteUint64 := F_WriteUInt64(THIS^.stCtx, nTmp);
END_METHOD

END_FUNCTION_BLOCK

// ---- RepeatedField/FB_RepeatedField.TcPOU
// Generic wrapper for ARRAY[*] OF T
FUNCTION_BLOCK FINAL FB_RepeatedField IMPLEMENTS I_RepeatedField
VAR_INPUT
END_VAR
VAR_OUTPUT
END_VAR
VAR
	anyArrayField       : T_Any;
    anyFirstElemField   : T_Any;
    ipFieldCodecField	: I_FieldCodec;
END_VAR
VAR
	nCapacityField		: UDINT;
	nCountField			: UDINT;		// Actual number of elements in the Array
END_VAR

// Adds the entries from the given parse context, decoding them with the specified codec.
METHOD AddEntriesFrom : HRESULT
VAR_IN_OUT CONSTANT
	fbParseCtx	: FB_ParseContext;
END_VAR
VAR_INPUT
	ipFieldCodec : I_FieldCodec;
END_VAR
VAR_OUTPUT
	nCount : UDINT;
END_VAR
VAR
	refCtx	: REFERENCE TO ST_ParseContext;
END_VAR
refCtx REF= fbParseCtx.refCtx;
THIS^.ipFieldCodecField := ipFieldCodec;
AddEntriesFrom := F_ReadRepeatedField(stCtx:= refCtx, ipRepeatedField:= THIS^, nLength=> nCount);
END_METHOD

METHOD CalculatePackedDataSize : HRESULT
VAR_OUTPUT
    nPackedDataSize : UDINT;
END_VAR
IF ipFieldCodecField = NULL OR THIS^.anyFirstElemField.pValue = NULL THEN
	CalculatePackedDataSize := E_WriterErrorCode.InternalError;
	RETURN;
END_IF

IF THIS^.nCountField = 0 THEN
	nPackedDataSize := 0;
	RETURN;
END_IF 

CalculatePackedDataSize := ipFieldCodecField.CalculatePackedDataSize(
								anyFirstElem:= THIS^.anyFirstElemField,
								nLength:= THIS^.nCount,
								nPackedDataSize=> nPackedDataSize);
END_METHOD

METHOD CalculateSize : HRESULT
VAR_OUTPUT
	nSize : UDINT;
END_VAR
VAR
	nPackedSize : UDINT;
END_VAR
IF ipFieldCodecField = NULL OR THIS^.anyFirstElemField.pValue = NULL THEN
	CalculateSize := E_WriterErrorCode.InternalError;
	RETURN;
END_IF

IF THIS^.nCountField = 0 THEN
	nSize := 0;
	RETURN;
END_IF

IF ipFieldCodecField.IsPackedRepeatedField(ipFieldCodecField.Tag) THEN
	
	CalculateSize := CalculatePackedDataSize(nPackedDataSize=> nPackedSize);
	IF FAILED(CalculateSize) THEN
		RETURN;
	END_IF
	nSize := F_ComputeRawVarint32Size(ipFieldCodecField.Tag) + F_ComputeLengthSize(nPackedSize) + nPackedSize;
    RETURN;
END_IF

CalculateSize := CalculatePackedDataSize(nPackedDataSize=> nPackedSize);
IF FAILED(CalculateSize) THEN
	RETURN;
END_IF

nSize := (F_ComputeRawVarint32Size(ipFieldCodecField.Tag) * THIS^.nCountField) + nPackedSize;
IF ipFieldCodecField.EndTag <> 0 THEN
	nSize := nSize + (F_ComputeRawVarint32Size(ipFieldCodecField.EndTag) * THIS^.nCountField);
END_IF
END_METHOD

METHOD PRIVATE ComputeCapacity : UDINT
VAR_INPUT
END_VAR
VAR
	nTotalSize		: UDINT;
	nElementSize	: UDINT;
END_VAR

nTotalSize := TO_UDINT(anyArrayField.diSize);
IF nTotalSize = 0 THEN
	RETURN;
END_IF

nElementSize := TO_UDINT(anyFirstElemField.diSize);
IF nElementSize = 0 THEN
	RETURN;
END_IF

ComputeCapacity := nTotalSize / nElementSize;
END_METHOD

METHOD ElementAtIndex : T_ANY
VAR_INPUT
	nIndex	: UDINT;
END_VAR
ElementAtIndex := THIS^.anyFirstElemField;

IF nIndex > nCapacityField - 1 THEN
	RETURN;
END_IF

ElementAtIndex := THIS^.anyFirstElemField;
ElementAtIndex.pValue := THIS^.anyFirstElemField.pValue + (nIndex * TO_UDINT(THIS^.anyFirstElemField.diSize));
END_METHOD

//FB_Init is always available implicitly and it is used primarily for initialization.
//The return value is not evaluated. For a specific influence, you can also declare the
//methods explicitly and provide additional code there with the standard initialization
//code. You can evaluate the return value.
METHOD FB_Init: BOOL
VAR_INPUT
    bInitRetains: BOOL; // TRUE: the retain variables are initialized (reset warm / reset cold)
    bInCopyCode: BOOL;  // TRUE: the instance will be copied to the copy code afterward (online change)   
	anyArray        : T_Any;
    anyFirstElem    : T_Any;
END_VAR
anyArrayField       := anyArray;
anyFirstElemField   := anyFirstElem;

Initialize();
END_METHOD

METHOD Initialize : HRESULT
VAR_INPUT
END_VAR

nCapacityField := ComputeCapacity();
nCountField 	:= 0;
END_METHOD

METHOD InitializeFromArray : HRESULT
VAR_INPUT
	anyArray        : T_Any;
    anyFirstElem    : T_Any;
	nCount			: UDINT;
END_VAR
anyArrayField       := anyArray;
anyFirstElemField   := anyFirstElem;

Initialize();
IF nCount <= THIS^.nCapacityField THEN
	THIS^.nCountField := nCount;
END_IF
END_METHOD

PROPERTY ipFieldCodec : I_FieldCodec
GET
ipFieldCodec := ipFieldCodecField;
END_GET
END_PROPERTY

PROPERTY nCapcacity : UDINT
GET
nCapcacity := nCapacityField;
END_GET
END_PROPERTY

PROPERTY nCount : UDINT
GET
nCount := THIS^.nCountField;
END_GET
SET
THIS^.nCountField := MIN(nCount, THIS^.nCapacityField);
END_SET
END_PROPERTY

// Sets the given value at the current element and increases nCount
METHOD SetValue : HRESULT
VAR_INPUT
	anyValue	: T_ANY;
END_VAR
VAR
	anyCurrentElem : T_ANY;
END_VAR

IF THIS^.nCountField > THIS^.nCapacityField THEN
	SetValue := E_ParserErrorCode.NotEnoughMem;
	RETURN;
END_IF

anyCurrentElem := THIS^.ElementAtIndex(THIS^.nCountField);

MEMCPY(destAddr:= anyCurrentElem.pValue, srcAddr:= anyValue.pValue, n:= TO_UDINT(MIN(anyCurrentElem.diSize, anyValue.diSize)));
 
THIS^.nCountField := THIS^.nCountField + 1;
END_METHOD

// Writes the contents of this collection to the given write context, encoding each
// value using the specified codec.
METHOD WriteTo : HRESULT
VAR_IN_OUT CONSTANT
	fbWriteCtx	: FB_WriteContext;
END_VAR
VAR_INPUT
	ipFieldCodec : I_FieldCodec;
END_VAR
VAR
	refCtx	: REFERENCE TO ST_WriteContext;
END_VAR
refCtx REF= fbWriteCtx.refCtx;
THIS^.ipFieldCodecField := ipFieldCodec;
WriteTo := F_WriteRepeatedField(stCtx:= refCtx, ipRepeatedField:= THIS^);
END_METHOD

// Writes the contents of this collection to the given write context, encoding each
// value using the specified codec.
METHOD WriteToWithCount : HRESULT
VAR_IN_OUT CONSTANT
	fbWriteCtx	: FB_WriteContext;
END_VAR
VAR_INPUT
	ipFieldCodec : I_FieldCodec;
	nCount		 : UDINT;			// Number of items in the collection.
END_VAR

THIS^.nCount := nCount;
WriteToWithCount := WriteTo(fbWriteCtx, ipFieldCodec);
END_METHOD

END_FUNCTION_BLOCK

// ---- RepeatedField/F_ReadRepeatedField.TcPOU
FUNCTION INTERNAL F_ReadRepeatedField : HRESULT
VAR_IN_OUT      
    stCtx : ST_ParseContext;
END_VAR
VAR_INPUT CONSTANT
	ipRepeatedField	: I_RepeatedField;
END_VAR
VAR_OUTPUT
	nLength : UDINT;
END_VAR
VAR
	nLastTag		: UDINT;
    hr          	: HRESULT;
    nCurrentLimit 	: UDINT;
    bTagConsumed	: BOOL;
    nBufferEnd  	: UDINT;  
    anyValue        : T_Any;
END_VAR

nLength := 0;

IF ipRepeatedField.ipFieldCodec = 0 THEN
    F_ReadRepeatedField := F_ParseError(stCtx,  E_ParserErrorCode.InternalError);
    RETURN;
END_IF

IF ipRepeatedField.nCapcacity = 0 THEN
    nLength := ipRepeatedField.nCount;
	RETURN;
END_IF

nLastTag := stCtx.stState.nLastTag;

IF ipRepeatedField.ipFieldCodec.IsPackedRepeatedField(nLastTag) THEN
    
    hr := F_ParseLength(stCtx, nLength=> nLength);
    IF FAILED(hr) OR nLength <= 0 THEN
        // Empty packed field, valid - ignore.
        F_ReadRepeatedField := hr;
        nLength := ipRepeatedField.nCount;
        RETURN;
    END_IF 
    
    F_SbhPushLimit(stCtx.stState, nLength, nCurrentLimit=> nCurrentLimit);
    nBufferEnd := stCtx.stState.nBufferPos + nLength;
    WHILE NOT F_SbhIsReachedLimit(stCtx.stState) DO
        hr := ipRepeatedField.ipFieldCodec.ValueReader(stCtx, anyOut=> anyValue);
        IF FAILED(hr) THEN
            F_ReadRepeatedField := hr;
            RETURN;
        END_IF
        
		hr := ipRepeatedField.SetValue(anyValue);
		IF FAILED(hr) THEN
            F_ReadRepeatedField := hr;
            RETURN;
        END_IF
    END_WHILE

    F_SbhPopLimit(stCtx.stState, nCurrentLimit);
ELSE
    // Not packed or possibly not packable...
    REPEAT
        hr := ipRepeatedField.ipFieldCodec.ValueReader(stCtx, anyOut=> anyValue);
        IF FAILED(hr) THEN
            F_ReadRepeatedField := hr;
            RETURN;
        END_IF
        
		hr := ipRepeatedField.SetValue(anyValue);
		IF FAILED(hr) THEN
            F_ReadRepeatedField := hr;
            RETURN;
        END_IF
        
        hr := F_MaybeConsumeTag(stCtx, nLastTag, bConsumed=> bTagConsumed);
        IF FAILED(hr) THEN
            F_ReadRepeatedField := hr;
            RETURN;
        END_IF
    UNTIL
        NOT bTagConsumed
    END_REPEAT
END_IF

nLength := ipRepeatedField.nCount;

END_FUNCTION

// ---- __TESTs/EnumTests/FB_ComputeEnumSizeTests.TcPOU
FUNCTION_BLOCK INTERNAL FINAL FB_ComputeEnumSizeTests EXTENDS FB_TestSuite
VAR_INPUT
END_VAR
VAR_OUTPUT
END_VAR
VAR
END_VAR

ShouldComputeByteBackedEnumSizeFromOwnStorageOnly();
ShouldComputeWordBackedEnumSizeFromOwnStorageOnly();
ShouldComputeDwordBackedEnumSize();
ShouldReturnZeroForNonEnum();

METHOD PRIVATE ShouldComputeByteBackedEnumSizeFromOwnStorageOnly : REFERENCE TO FB_Test
VAR
    aValues : ARRAY[0..3] OF E_DataType := [
        E_DataType.DATA_TYPE_HUMIDITY,
        E_DataType.DATA_TYPE_PRESSURE,
        E_DataType.DATA_TYPE_TEMPERATURE,
        E_DataType.DATA_TYPE_UNKNOWN];
    nActual : UDINT;
END_VAR
TEST(__POUNAME());

nActual := F_ComputeEnumSize(anyEnum:= aValues[0]);

AssertEquals_UDINT(
    Expected:= 1,
    Actual:= nActual,
    Message:= 'Expected BYTE backed enum size to use only the enum storage');

TEST_FINISHED_NAMED(__POUNAME());
END_METHOD

METHOD PRIVATE ShouldComputeDwordBackedEnumSize : REFERENCE TO FB_Test
VAR
    eValue : E_Status := E_Status.STATUS_ERROR;
    nActual : UDINT;
END_VAR
TEST(__POUNAME());

nActual := F_ComputeEnumSize(anyEnum:= eValue);

AssertEquals_UDINT(
    Expected:= 1,
    Actual:= nActual,
    Message:= 'Expected DWORD backed enum size to match its varint size');

TEST_FINISHED_NAMED(__POUNAME());
END_METHOD

METHOD PRIVATE ShouldComputeWordBackedEnumSizeFromOwnStorageOnly : REFERENCE TO FB_Test
VAR
    aValues : ARRAY[0..1] OF E_Color := [
        E_Color.COLOR_BLUE,
        E_Color.COLOR_GREEN];
    nActual : UDINT;
END_VAR
TEST(__POUNAME());

nActual := F_ComputeEnumSize(anyEnum:= aValues[0]);

AssertEquals_UDINT(
    Expected:= 1,
    Actual:= nActual,
    Message:= 'Expected WORD backed enum size to use only the enum storage');

TEST_FINISHED_NAMED(__POUNAME());
END_METHOD

METHOD PRIVATE ShouldReturnZeroForNonEnum : REFERENCE TO FB_Test
VAR
    nValue : UDINT := 3;
    nActual : UDINT;
END_VAR
TEST(__POUNAME());

nActual := F_ComputeEnumSize(anyEnum:= nValue);

AssertEquals_UDINT(
    Expected:= 0,
    Actual:= nActual,
    Message:= 'Expected non-enum input to have size 0');

TEST_FINISHED_NAMED(__POUNAME());
END_METHOD

END_FUNCTION_BLOCK

// ---- __TESTs/EnumTests/FB_FieldCodecEnumTests.TcPOU
FUNCTION_BLOCK INTERNAL FINAL FB_FieldCodecEnumTests EXTENDS FB_TestSuite
VAR_INPUT
END_VAR
VAR_OUTPUT
END_VAR
VAR
    fbFieldCodec : FB_FieldCodecEnum(nTag:= 0);
END_VAR

ShouldCalculatePackedSizeFromEnumStorageOnly();
ShouldWriteEnumValuesFromEnumStorageOnly();
ShouldReadEnumValueForRepeatedFieldStorage();

METHOD PRIVATE ShouldCalculatePackedSizeFromEnumStorageOnly : REFERENCE TO FB_Test
VAR
    aValues : ARRAY[0..1] OF E_Color := [
        E_Color.COLOR_BLUE,
        E_Color.COLOR_GREEN];
    nPackedDataSize : UDINT;
    hrActual : HRESULT;
END_VAR
TEST(__POUNAME());

hrActual := fbFieldCodec.CalculatePackedDataSize(
    anyFirstElem:= F_ToAnyType(aValues[0]),
    nLength:= 2,
    nPackedDataSize=> nPackedDataSize);

AssertEquals_DINT(
    Expected:= S_OK,
    Actual:= hrActual,
    Message:= 'Expected enum packed size calculation to succeed');

AssertEquals_UDINT(
    Expected:= 2,
    Actual:= nPackedDataSize,
    Message:= 'Expected packed size to use only the enum storage for each item');

TEST_FINISHED_NAMED(__POUNAME());
END_METHOD

METHOD PRIVATE ShouldReadEnumValueForRepeatedFieldStorage : REFERENCE TO FB_Test
VAR_INST
    fbCtx : FB_ParseContext;
END_VAR
VAR
    cBuffer : ARRAY[0..7] OF BYTE := [16#03];
    refCtx : REFERENCE TO ST_ParseContext;
    anyOut : T_Any;
    nActual : UDINT;
    hrActual : HRESULT;
END_VAR
TEST(__POUNAME());

fbCtx.FromBuffer(cBuffer);
refCtx REF= fbCtx.refCtx;

hrActual := fbFieldCodec.ValueReader(stCtx:= refCtx, anyOut=> anyOut);
IF SUCCEEDED(hrActual) THEN
    MEMCPY(destAddr:= ADR(nActual), srcAddr:= anyOut.pValue, n:= MIN(TO_UDINT(anyOut.diSize), SIZEOF(nActual)));
END_IF

AssertEquals_DINT(
    Expected:= S_OK,
    Actual:= hrActual,
    Message:= 'Expected enum codec reader to parse a varint enum value');

AssertEquals_UDINT(
    Expected:= 3,
    Actual:= nActual,
    Message:= 'Expected parsed enum value 3');

AssertEquals_UDINT(
    Expected:= 1,
    Actual:= fbCtx.refCtx.stState.nBufferPos,
    Message:= 'Expected read position after one-byte enum value');

TEST_FINISHED_NAMED(__POUNAME());
END_METHOD

METHOD PRIVATE ShouldWriteEnumValuesFromEnumStorageOnly : REFERENCE TO FB_Test
VAR_INST
    fbCtx : FB_WriteContext;
END_VAR
VAR
    cExpectedBuffer : ARRAY[0..7] OF BYTE := [16#03, 16#03, 16#02];
    aDataTypes : ARRAY[0..1] OF E_DataType := [
        E_DataType.DATA_TYPE_HUMIDITY,
        E_DataType.DATA_TYPE_PRESSURE];
    aColors : ARRAY[0..1] OF E_Color := [
        E_Color.COLOR_BLUE,
        E_Color.COLOR_GREEN];
    eStatus : E_Status := E_Status.STATUS_ERROR;
    aActualBuffer : ARRAY[0..7] OF BYTE;
    refCtx : REFERENCE TO ST_WriteContext;
    hrActual : HRESULT;
END_VAR
TEST(__POUNAME());

fbCtx.FromBuffer(aActualBuffer);
refCtx REF= fbCtx.refCtx;

hrActual := fbFieldCodec.ValueWriter(stCtx:= refCtx, anyIn:= F_ToAnyType(aDataTypes[0]));
IF SUCCEEDED(hrActual) THEN
    hrActual := fbFieldCodec.ValueWriter(stCtx:= refCtx, anyIn:= F_ToAnyType(aColors[0]));
END_IF
IF SUCCEEDED(hrActual) THEN
    hrActual := fbFieldCodec.ValueWriter(stCtx:= refCtx, anyIn:= F_ToAnyType(eStatus));
END_IF

AssertEquals_DINT(
    Expected:= S_OK,
    Actual:= hrActual,
    Message:= 'Expected enum codec writer to accept BYTE, WORD and DWORD backed enums');

AssertArrayEquals_BYTE(
    Expecteds:= cExpectedBuffer,
    Actuals:= aActualBuffer,
    Message:= 'Expected enum values to be written as value 3 without reading neighbour storage');

AssertEquals_UDINT(
    Expected:= 3,
    Actual:= fbCtx.refCtx.stState.nBufferPos,
    Message:= 'Expected write position after three one-byte enum values');

TEST_FINISHED_NAMED(__POUNAME());
END_METHOD

END_FUNCTION_BLOCK

// ---- __TESTs/EnumTests/FB_ReadEnumTests.TcPOU
FUNCTION_BLOCK INTERNAL FINAL FB_ReadEnumTests EXTENDS FB_TestSuite
VAR_INPUT
END_VAR
VAR_OUTPUT
END_VAR
VAR
END_VAR

ShouldReadByteBackedEnumWithoutChangingNeighbourValues();
ShouldReadWordBackedEnumWithoutChangingNeighbourValues();
ShouldReadDwordBackedEnum();
ShouldReturnInvalidDataForNonEnum();

METHOD PRIVATE ShouldReadByteBackedEnumWithoutChangingNeighbourValues : REFERENCE TO FB_Test
VAR_INST
    fbCtx : FB_ParseContext;
END_VAR
VAR
    cBuffer : ARRAY[0..7] OF BYTE := [16#03];
    aValues : ARRAY[0..3] OF E_DataType := [
        E_DataType.DATA_TYPE_UNKNOWN,
        E_DataType.DATA_TYPE_TEMPERATURE,
        E_DataType.DATA_TYPE_PRESSURE,
        E_DataType.DATA_TYPE_HUMIDITY];
    nActual : BYTE;
    nNeighbour : BYTE;
    hrActual : HRESULT;
END_VAR
TEST(__POUNAME());

fbCtx.FromBuffer(cBuffer);

hrActual := fbCtx.ReadEnum(anyEnum:= aValues[0]);
MEMCPY(destAddr:= ADR(nActual), srcAddr:= ADR(aValues[0]), n:= SIZEOF(nActual));
MEMCPY(destAddr:= ADR(nNeighbour), srcAddr:= ADR(aValues[1]), n:= SIZEOF(nNeighbour));

AssertEquals_DINT(
    Expected:= S_OK,
    Actual:= hrActual,
    Message:= 'Expected S_OK when reading BYTE backed enum');

AssertEquals_UDINT(
    Expected:= 3,
    Actual:= TO_UDINT(nActual),
    Message:= 'Expected BYTE backed enum value 3');

AssertEquals_UDINT(
    Expected:= 1,
    Actual:= TO_UDINT(nNeighbour),
    Message:= 'Expected neighbouring BYTE backed enum value to stay unchanged');

AssertEquals_UDINT(
    Expected:= 1,
    Actual:= fbCtx.refCtx.stState.nBufferPos,
    Message:= 'Expected read position after one-byte enum value');

TEST_FINISHED_NAMED(__POUNAME());
END_METHOD

METHOD PRIVATE ShouldReadDwordBackedEnum : REFERENCE TO FB_Test
VAR_INST
    fbCtx : FB_ParseContext;
END_VAR
VAR
    cBuffer : ARRAY[0..7] OF BYTE := [16#02];
    eValue : E_Status := E_Status.STATUS_IDLE;
    nActual : DWORD;
    hrActual : HRESULT;
END_VAR
TEST(__POUNAME());

fbCtx.FromBuffer(cBuffer);

hrActual := fbCtx.ReadEnum(anyEnum:= eValue);
MEMCPY(destAddr:= ADR(nActual), srcAddr:= ADR(eValue), n:= SIZEOF(nActual));

AssertEquals_DINT(
    Expected:= S_OK,
    Actual:= hrActual,
    Message:= 'Expected S_OK when reading DWORD backed enum');

AssertEquals_UDINT(
    Expected:= 2,
    Actual:= TO_UDINT(nActual),
    Message:= 'Expected DWORD backed enum value 2');

AssertEquals_UDINT(
    Expected:= 1,
    Actual:= fbCtx.refCtx.stState.nBufferPos,
    Message:= 'Expected read position after one-byte enum value');

TEST_FINISHED_NAMED(__POUNAME());
END_METHOD

METHOD PRIVATE ShouldReadWordBackedEnumWithoutChangingNeighbourValues : REFERENCE TO FB_Test
VAR_INST
    fbCtx : FB_ParseContext;
END_VAR
VAR
    cBuffer : ARRAY[0..7] OF BYTE := [16#03];
    aValues : ARRAY[0..1] OF E_Color := [
        E_Color.COLOR_DEFAULT,
        E_Color.COLOR_RED];
    nActual : WORD;
    nNeighbour : WORD;
    hrActual : HRESULT;
END_VAR
TEST(__POUNAME());

fbCtx.FromBuffer(cBuffer);

hrActual := fbCtx.ReadEnum(anyEnum:= aValues[0]);
MEMCPY(destAddr:= ADR(nActual), srcAddr:= ADR(aValues[0]), n:= SIZEOF(nActual));
MEMCPY(destAddr:= ADR(nNeighbour), srcAddr:= ADR(aValues[1]), n:= SIZEOF(nNeighbour));

AssertEquals_DINT(
    Expected:= S_OK,
    Actual:= hrActual,
    Message:= 'Expected S_OK when reading WORD backed enum');

AssertEquals_UDINT(
    Expected:= 3,
    Actual:= TO_UDINT(nActual),
    Message:= 'Expected WORD backed enum value 3');

AssertEquals_UDINT(
    Expected:= 1,
    Actual:= TO_UDINT(nNeighbour),
    Message:= 'Expected neighbouring WORD backed enum value to stay unchanged');

AssertEquals_UDINT(
    Expected:= 1,
    Actual:= fbCtx.refCtx.stState.nBufferPos,
    Message:= 'Expected read position after one-byte enum value');

TEST_FINISHED_NAMED(__POUNAME());
END_METHOD

METHOD PRIVATE ShouldReturnInvalidDataForNonEnum : REFERENCE TO FB_Test
VAR_INST
    fbCtx : FB_ParseContext;
END_VAR
VAR
    cBuffer : ARRAY[0..7] OF BYTE := [16#03];
    nValue : UDINT;
    hrExpected : HRESULT := E_HRESULTAdsErr.INVALIDDATA;
    hrActual : HRESULT;
END_VAR
TEST(__POUNAME());

fbCtx.FromBuffer(cBuffer);

hrActual := fbCtx.ReadEnum(anyEnum:= nValue);

AssertEquals_DINT(
    Expected:= hrExpected,
    Actual:= hrActual,
    Message:= 'Expected INVALIDDATA for non-enum input');

AssertEquals_UDINT(
    Expected:= 0,
    Actual:= fbCtx.refCtx.stState.nBufferPos,
    Message:= 'Expected read position to stay unchanged');

TEST_FINISHED_NAMED(__POUNAME());
END_METHOD

END_FUNCTION_BLOCK

// ---- __TESTs/EnumTests/FB_WriteEnumTests.TcPOU
FUNCTION_BLOCK INTERNAL FINAL FB_WriteEnumTests EXTENDS FB_TestSuite
VAR_INPUT
END_VAR
VAR_OUTPUT
END_VAR
VAR
END_VAR

ShouldWriteByteBackedEnumFromOwnStorageOnly();
ShouldWriteWordBackedEnumFromOwnStorageOnly();
ShouldWriteDwordBackedEnum();
ShouldReturnInvalidDataForNonEnum();

METHOD PRIVATE ShouldReturnInvalidDataForNonEnum : REFERENCE TO FB_Test
VAR_INST
    fbCtx : FB_WriteContext;
END_VAR
VAR
    aActualBuffer : ARRAY[0..7] OF BYTE;
    nValue : UDINT := 3;
    hrExpected : HRESULT := E_HRESULTAdsErr.INVALIDDATA;
    hrActual : HRESULT;
END_VAR
TEST(__POUNAME());

fbCtx.FromBuffer(aActualBuffer);

hrActual := fbCtx.WriteEnum(anyEnum:= nValue);

AssertEquals_DINT(
    Expected:= hrExpected,
    Actual:= hrActual,
    Message:= 'Expected INVALIDDATA for non-enum input');

AssertEquals_UDINT(
    Expected:= 0,
    Actual:= fbCtx.refCtx.stState.nBufferPos,
    Message:= 'Expected write position to stay unchanged');

TEST_FINISHED_NAMED(__POUNAME());
END_METHOD

METHOD PRIVATE ShouldWriteByteBackedEnumFromOwnStorageOnly : REFERENCE TO FB_Test
VAR_INST
    fbCtx : FB_WriteContext;
END_VAR
VAR
    cExpectedBuffer : ARRAY[0..7] OF BYTE := [16#03];
    aValues : ARRAY[0..3] OF E_DataType := [
        E_DataType.DATA_TYPE_HUMIDITY,
        E_DataType.DATA_TYPE_PRESSURE,
        E_DataType.DATA_TYPE_TEMPERATURE,
        E_DataType.DATA_TYPE_UNKNOWN];
    aActualBuffer : ARRAY[0..7] OF BYTE;
    hrActual : HRESULT;
END_VAR
TEST(__POUNAME());

fbCtx.FromBuffer(aActualBuffer);

hrActual := fbCtx.WriteEnum(anyEnum:= aValues[0]);

AssertEquals_DINT(
    Expected:= S_OK,
    Actual:= hrActual,
    Message:= 'Expected S_OK when writing BYTE backed enum');

AssertArrayEquals_BYTE(
    Expecteds:= cExpectedBuffer,
    Actuals:= aActualBuffer,
    Message:= 'Expected BYTE backed enum to be written as value 3 only');

AssertEquals_UDINT(
    Expected:= 1,
    Actual:= fbCtx.refCtx.stState.nBufferPos,
    Message:= 'Expected write position after one-byte enum value');

TEST_FINISHED_NAMED(__POUNAME());
END_METHOD

METHOD PRIVATE ShouldWriteDwordBackedEnum : REFERENCE TO FB_Test
VAR_INST
    fbCtx : FB_WriteContext;
END_VAR
VAR
    cExpectedBuffer : ARRAY[0..7] OF BYTE := [16#02];
    eValue : E_Status := E_Status.STATUS_ERROR;
    aActualBuffer : ARRAY[0..7] OF BYTE;
    hrActual : HRESULT;
END_VAR
TEST(__POUNAME());

fbCtx.FromBuffer(aActualBuffer);

hrActual := fbCtx.WriteEnum(anyEnum:= eValue);

AssertEquals_DINT(
    Expected:= S_OK,
    Actual:= hrActual,
    Message:= 'Expected S_OK when writing DWORD backed enum');

AssertArrayEquals_BYTE(
    Expecteds:= cExpectedBuffer,
    Actuals:= aActualBuffer,
    Message:= 'Expected DWORD backed enum to be written as value 2');

AssertEquals_UDINT(
    Expected:= 1,
    Actual:= fbCtx.refCtx.stState.nBufferPos,
    Message:= 'Expected write position after one-byte enum value');

TEST_FINISHED_NAMED(__POUNAME());
END_METHOD

METHOD PRIVATE ShouldWriteWordBackedEnumFromOwnStorageOnly : REFERENCE TO FB_Test
VAR_INST
    fbCtx : FB_WriteContext;
END_VAR
VAR
    cExpectedBuffer : ARRAY[0..7] OF BYTE := [16#03];
    aValues : ARRAY[0..1] OF E_Color := [
        E_Color.COLOR_BLUE,
        E_Color.COLOR_GREEN];
    aActualBuffer : ARRAY[0..7] OF BYTE;
    hrActual : HRESULT;
END_VAR
TEST(__POUNAME());

fbCtx.FromBuffer(aActualBuffer);

hrActual := fbCtx.WriteEnum(anyEnum:= aValues[0]);

AssertEquals_DINT(
    Expected:= S_OK,
    Actual:= hrActual,
    Message:= 'Expected S_OK when writing WORD backed enum');

AssertArrayEquals_BYTE(
    Expecteds:= cExpectedBuffer,
    Actuals:= aActualBuffer,
    Message:= 'Expected WORD backed enum to be written as value 3 only');

AssertEquals_UDINT(
    Expected:= 1,
    Actual:= fbCtx.refCtx.stState.nBufferPos,
    Message:= 'Expected write position after one-byte enum value');

TEST_FINISHED_NAMED(__POUNAME());
END_METHOD

END_FUNCTION_BLOCK

// ---- __TESTs/EnumTests/PRG_EnumTests.TcPOU
{attribute 'analysis' := '-33'}
PROGRAM INTERNAL PRG_EnumTests
VAR
{IF defined (UNIT_TEST)}
    fbComputeEnumSizeTests : FB_ComputeEnumSizeTests;
    fbWriteEnumTests       : FB_WriteEnumTests;
    fbReadEnumTests        : FB_ReadEnumTests;
    fbFieldCodecEnumTests  : FB_FieldCodecEnumTests;
{END_IF}
END_VAR

END_PROGRAM

// ---- __TESTs/MessagesTests/POUs/FB_ReadMessageErrorTests.TcPOU
FUNCTION_BLOCK INTERNAL FINAL FB_ReadMessageErrorTests EXTENDS FB_TestSuite
VAR
    fbMessage : FB_TestFixed32Message;
END_VAR

ShouldPreserveRawMessageFailure();

METHOD PRIVATE ShouldPreserveRawMessageFailure : REFERENCE TO FB_Test
VAR CONSTANT
    cBuffer : ARRAY[0..1] OF BYTE := [16#01, 16#0D];
END_VAR
VAR_INST
    fbCtx : FB_ParseContext;
END_VAR
VAR
    hr : HRESULT;
END_VAR
TEST(__POUNAME());

fbCtx.FromBuffer(cBuffer);

hr := F_ReadMessage(fbCtx:= fbCtx, iMessage:= fbMessage);

AssertEquals_DINT(
    Expected:= E_ParserErrorCode.TruncatedMessage,
    Actual:= hr,
    Message:= 'Expected F_ReadMessage to preserve the original raw message error');

AssertEquals_DINT(
    Expected:= E_ParserErrorCode.TruncatedMessage,
    Actual:= fbCtx.refCtx.stState.eParserErrorCode,
    Message:= 'Expected parser state to keep the original raw message error');

TEST_FINISHED_NAMED(__POUNAME());
END_METHOD

END_FUNCTION_BLOCK

// ---- __TESTs/RepeatedFieldTests/FB_TestFixed32Message.TcPOU
FUNCTION_BLOCK INTERNAL FINAL FB_TestFixed32Message IMPLEMENTS I_Message
VAR
    fbMessageParser : FB_MessageParser(ipMessage:= THIS^);
    fbMessageWriter : FB_MessageWriter(ipMessage:= THIS^);
    nValue : UDINT;
END_VAR

METHOD CalculateSize : UDINT
VAR_INPUT
END_VAR
CalculateSize := F_ComputeTagSize(1) + SIZEOF(nValue);
END_METHOD

METHOD MergeFrom : HRESULT
VAR_IN_OUT
    fbParseCtx : FB_ParseContext;
END_VAR
VAR
    nTag : UDINT;
END_VAR
REPEAT
MergeFrom := fbParseCtx.ReadTag(nTag=> nTag);
IF SUCCEEDED(MergeFrom) AND nTag = 0 THEN
    EXIT;
END_IF

IF FAILED(MergeFrom) THEN
    RETURN;
END_IF

CASE nTag OF
    16#0D:
        MergeFrom := fbParseCtx.ReadFixed32(nValue=> nValue);
ELSE
    MergeFrom := fbParseCtx.SkipLastField();
END_CASE
UNTIL FAILED(MergeFrom) OR nTag = 0
END_REPEAT
END_METHOD

PROPERTY MessageValue : T_Any
GET
MessageValue := F_ToAnyType(anyArg:= nValue);
END_GET
END_PROPERTY

PROPERTY Parser : REFERENCE TO FB_MessageParser
GET
Parser REF= fbMessageParser;
END_GET
END_PROPERTY

PROPERTY Writer : REFERENCE TO FB_MessageWriter
GET
Writer REF= fbMessageWriter;
END_GET
END_PROPERTY

METHOD WriteTo : HRESULT
VAR_IN_OUT
    fbWriteCtx : FB_WriteContext;
END_VAR
WriteTo := fbWriteCtx.WriteTag(1, E_WireType.Fixed32);
IF FAILED(WriteTo) THEN
    RETURN;
END_IF

WriteTo := fbWriteCtx.WriteFixed32(nValue);
END_METHOD

END_FUNCTION_BLOCK

// ---- __TESTs/MessagesTests/POUs/FB_TestWrongSizeMessage.TcPOU
FUNCTION_BLOCK INTERNAL FINAL FB_TestWrongSizeMessage IMPLEMENTS I_Message
VAR
    fbMessageParser : FB_MessageParser(ipMessage:= THIS^);
    fbMessageWriter : FB_MessageWriter(ipMessage:= THIS^);
    nValue : UDINT := 16#12345678;
END_VAR

METHOD CalculateSize : UDINT
VAR_INPUT
END_VAR
CalculateSize := 0;
END_METHOD

METHOD MergeFrom : HRESULT
VAR_IN_OUT
    fbParseCtx : FB_ParseContext;
END_VAR
VAR
    nTag : UDINT;
END_VAR
REPEAT
MergeFrom := fbParseCtx.ReadTag(nTag=> nTag);
IF SUCCEEDED(MergeFrom) AND nTag = 0 THEN
    EXIT;
END_IF

IF FAILED(MergeFrom) THEN
    RETURN;
END_IF

CASE nTag OF
    16#0D:
        MergeFrom := fbParseCtx.ReadFixed32(nValue=> nValue);
ELSE
    MergeFrom := fbParseCtx.SkipLastField();
END_CASE
UNTIL FAILED(MergeFrom) OR nTag = 0
END_REPEAT
END_METHOD

PROPERTY MessageValue : T_Any
GET
MessageValue := F_ToAnyType(anyArg:= nValue);
END_GET
END_PROPERTY

PROPERTY Parser : REFERENCE TO FB_MessageParser
GET
Parser REF= fbMessageParser;
END_GET
END_PROPERTY

PROPERTY Writer : REFERENCE TO FB_MessageWriter
GET
Writer REF= fbMessageWriter;
END_GET
END_PROPERTY

METHOD WriteTo : HRESULT
VAR_IN_OUT
    fbWriteCtx : FB_WriteContext;
END_VAR
WriteTo := fbWriteCtx.WriteTag(1, E_WireType.Fixed32);
IF FAILED(WriteTo) THEN
    RETURN;
END_IF

WriteTo := fbWriteCtx.WriteFixed32(nValue);
END_METHOD

END_FUNCTION_BLOCK

// ---- __TESTs/MessagesTests/POUs/FB_WriteMessageSizeTests.TcPOU
FUNCTION_BLOCK INTERNAL FINAL FB_WriteMessageSizeTests EXTENDS FB_TestSuite
VAR
    fbMessage : FB_TestWrongSizeMessage;
END_VAR

ShouldWriteMeasuredMessageLength();
ShouldComputeMessageSizeFromSerializedBytes();
ShouldExposeBytesWritten();

METHOD PRIVATE ShouldWriteMeasuredMessageLength : REFERENCE TO FB_Test
VAR CONSTANT
    cExpected : ARRAY[0..5] OF BYTE := [16#05, 16#0D, 16#78, 16#56, 16#34, 16#12];
END_VAR
VAR_INST
    fbCtx : FB_WriteContext;
END_VAR
VAR
    aActual : ARRAY[0..5] OF BYTE;
    hr : HRESULT;
END_VAR
TEST(__POUNAME());

fbCtx.FromBuffer(aActual);

hr := fbCtx.WriteMessage(ipMessage:= fbMessage);

AssertEquals_DINT(
    Expected:= S_OK,
    Actual:= hr,
    Message:= 'Expected embedded message write to succeed');

AssertArrayEquals_BYTE(
    Expecteds:= cExpected,
    Actuals:= aActual,
    Message:= 'Expected length prefix to use serialized byte count, not CalculateSize');

AssertEquals_UDINT(
    Expected:= 6,
    Actual:= fbCtx.refCtx.stState.nBufferPos,
    Message:= 'Expected writer position to include length and payload');

TEST_FINISHED_NAMED(__POUNAME());
END_METHOD

METHOD PRIVATE ShouldComputeMessageSizeFromSerializedBytes : REFERENCE TO FB_Test
VAR
    nSize : UDINT;
END_VAR
TEST(__POUNAME());

nSize := F_ComputeMessageSize(iMessage:= fbMessage);

AssertEquals_UDINT(
    Expected:= 6,
    Actual:= nSize,
    Message:= 'Expected message size to be measured from serialized bytes');

TEST_FINISHED_NAMED(__POUNAME());
END_METHOD

METHOD PRIVATE ShouldExposeBytesWritten : REFERENCE TO FB_Test
VAR
    aBuffer : ARRAY[0..4] OF BYTE;
    hr : HRESULT;
END_VAR
TEST(__POUNAME());

hr := fbMessage.Writer.WriteTo(aBuffer);

AssertEquals_DINT(
    Expected:= S_OK,
    Actual:= hr,
    Message:= 'Expected raw message write to succeed');

AssertEquals_UDINT(
    Expected:= 5,
    Actual:= fbMessage.Writer.nBytesWritten,
    Message:= 'Expected writer to expose actual raw payload byte count');

TEST_FINISHED_NAMED(__POUNAME());
END_METHOD

END_FUNCTION_BLOCK

// ---- __TESTs/MessagesTests/PRG_MessageTests.TcPOU
{attribute 'analysis' := '-33'}
PROGRAM INTERNAL PRG_MessageTests
VAR
    {IF defined (UNIT_TEST)}
    fbMessageTests  : FB_MessageTests;
    //fbRepeatedStringMessageTests : FB_RepeatedStringMessageTests;
    fbfbb : FB_FooMessage;
    fbExam : FB_ExampleMessage;
    
    fbRoundTripMessageExampleTest : FB_RoundTripMessageExampleTest;
    fbReadMessageErrorTests : FB_ReadMessageErrorTests;
    fbWriteMessageSizeTests : FB_WriteMessageSizeTests;
    {END_IF}
END_VAR

END_PROGRAM

// ---- __TESTs/PRG_UnitTests.TcPOU
{attribute 'analysis' := '-33'}
PROGRAM INTERNAL PRG_UnitTests
VAR
{IF defined (UNIT_TEST)}

{END_IF}
// fbTestNestedMessage1 : FB_TestNestedMessage;
// fbTestNestedMessage2 : FB_TestNestedMessage;
fbMotor : FB_Motor;
fbMotorDec : FB_Motor;
fbcplx : FB_ComplexData;
fbcplxDec : FB_ComplexData;
fbDevice : FB_Device;
fbScalarSrc : FB_ScalarTypesTest;
fbScalarDst : FB_ScalarTypesTest;
aBuffer	: ARRAY[0..1023] OF BYTE;
aBuffer1	: ARRAY[0..1023] OF BYTE;

_profiler : Profiler;
profilerData  : PROFILERSTRUCT;
END_VAR

{IF defined (UNIT_TEST)}
PRG_ParsingPrimitiveTests();
PRG_RoundTripTests();
PRG_WritingPrimitiveTests();
PRG_MessageTests();
PRG_WireFormatTests();
PRG_RepeatedFieldTests();
PRG_HelperTests();
PRG_EnumTests();
PRG_SpanTests();
TcUnit.RUN();

{END_IF}
//  fbMotor.Writer.WriteTo(aBuffer);
//  fbMotorDec.Parser.ParseFrom(aBuffer);
// fbcplx.Writer.WriteTo(aBuffer1);
// fbcplxDec.Parser.ParseFrom(aBuffer1);
// fbTestNestedMessage1.Writer.WriteTo(aBuffer);
// fbTestNestedMessage2.Parser.ParseFrom(aBuffer);

_profiler(START:= TRUE, RESET:= TRUE);
fbScalarSrc.Writer.WriteTo(aBuffer);
fbScalarDst.Parser.ParseFrom(aBuffer);

_profiler(START:=FALSE, RESET:= TRUE, DATA=> profilerData);

END_PROGRAM

// ---- __TESTs/RepeatedFieldTests/Read/FB_ReadRepeatedFieldMessageTests.TcPOU
FUNCTION_BLOCK INTERNAL FINAL FB_ReadRepeatedFieldMessageTests EXTENDS FB_TestSuite
VAR
    aActual : ARRAY[0..2] OF UDINT;
    fbMessage : FB_TestFixed32Message;
    fbFieldCodec : FB_FieldCodecMessage(nTag:= 16#0A, ipMessage:= fbMessage);
    fbRepeatedField : FB_RepeatedField(anyArray:= F_ToAnyType(aActual), anyFirstElem:= F_ToAnyType(aActual[0]));
END_VAR

ShouldReadNonPackedMessagesAndReturnItemCount();

METHOD PRIVATE ShouldReadNonPackedMessagesAndReturnItemCount : REFERENCE TO FB_Test
VAR CONSTANT
    cBuffer : ARRAY[0..20] OF BYTE := [
        16#0A, 16#05, 16#0D, 16#2A, 16#00, 16#00, 16#00,
        16#0A, 16#05, 16#0D, 16#39, 16#1B, 16#00, 16#00,
        16#0A, 16#05, 16#0D, 16#39, 16#05, 16#00, 16#00];
    cExpected : ARRAY[0..2] OF UDINT := [42, 6969, 1337];
END_VAR
VAR_INST
    fbCtx : FB_ParseContext;
END_VAR
VAR
    hr : HRESULT;
    nTag : UDINT;
    nActualCount : UDINT;
END_VAR
TEST(__POUNAME());

fbRepeatedField.Initialize();
MEMSET(destAddr:= ADR(aActual), fillByte:= 16#0, n:= SIZEOF(aActual));
fbCtx.FromBuffer(cBuffer);

F_ParseTag(fbCtx.refCtx, nTag=> nTag);
hr := fbRepeatedField.AddEntriesFrom(fbParseCtx:= fbCtx, ipFieldCodec:= fbFieldCodec, nCount=> nActualCount);

AssertEquals_DINT(
    Expected:= S_OK,
    Actual:= hr,
    Message:= 'Expected repeated message read to succeed');

AssertArrayEquals_UDINT(
    Expecteds:= cExpected,
    Actuals:= aActual,
    Message:= 'Expected all message values to be copied into repeated storage');

AssertEquals_UDINT(
    Expected:= 3,
    Actual:= nActualCount,
    Message:= 'Expected AddEntriesFrom to return the total item count');

AssertEquals_UDINT(
    Expected:= 21,
    Actual:= fbCtx.refCtx.stState.nBufferPos,
    Message:= 'Expected parser to consume all repeated messages');

TEST_FINISHED_NAMED(__POUNAME());
END_METHOD

END_FUNCTION_BLOCK

// ---- __TESTs/RepeatedFieldTests/Read/PRG_ReadRepeatedFieldTests.TcPOU
{attribute 'analysis' := '-33'}
PROGRAM INTERNAL PRG_ReadRepeatedFieldTests
{IF defined (UNIT_TEST)}
	fbReadRepeatedFieldBoolTests    : FB_ReadRepeatedFieldBoolTests;
	fbReadRepeatedFieldBytesTests   : FB_ReadRepeatedFieldBytesTests;
    fbReadRepeatedFieldUint32Tests  : FB_ReadRepeatedFieldUint32Tests;
    fbReadRepeatedFieldFixed32Tests : FB_ReadRepeatedFieldFixed32Tests;
    fbReadRepeatedFieldFixed64Tests : FB_ReadRepeatedFieldFixed64Tests;
    fbReadRepeatedFieldStringTests  : FB_ReadRepeatedFieldStringTests;
    fbReadRepeatedFieldMessageTests : FB_ReadRepeatedFieldMessageTests;
{END_IF}

END_PROGRAM

// ---- __TESTs/RepeatedFieldTests/Write/FB_WriteRepeatedFieldMessageTests.TcPOU
FUNCTION_BLOCK INTERNAL FINAL FB_WriteRepeatedFieldMessageTests EXTENDS FB_TestSuite
VAR
    aValues : ARRAY[0..2] OF UDINT := [42, 6969, 1337];
    fbMessage : FB_TestFixed32Message;
    fbFieldCodec : FB_FieldCodecMessage(nTag:= 16#0A, ipMessage:= fbMessage);
    fbRepeatedField : FB_RepeatedField(anyArray:= F_ToAnyType(aValues), anyFirstElem:= F_ToAnyType(aValues[0]));
END_VAR

ShouldWriteNonPackedMessagesAndCalculateSize();

METHOD PRIVATE ShouldWriteNonPackedMessagesAndCalculateSize : REFERENCE TO FB_Test
VAR CONSTANT
    cExpected : ARRAY[0..20] OF BYTE := [
        16#0A, 16#05, 16#0D, 16#2A, 16#00, 16#00, 16#00,
        16#0A, 16#05, 16#0D, 16#39, 16#1B, 16#00, 16#00,
        16#0A, 16#05, 16#0D, 16#39, 16#05, 16#00, 16#00];
END_VAR
VAR_INST
    fbCtx : FB_WriteContext;
END_VAR
VAR
    aActual : ARRAY[0..20] OF BYTE;
    hr : HRESULT;
    hrSize : HRESULT;
    nSize : UDINT;
END_VAR
TEST(__POUNAME());

fbRepeatedField.InitializeFromArray(anyArray:= F_ToAnyType(aValues), anyFirstElem:= F_ToAnyType(aValues[0]), nCount:= 3);
fbCtx.FromBuffer(aActual);

hr := fbRepeatedField.WriteToWithCount(fbWriteCtx:= fbCtx, ipFieldCodec:= fbFieldCodec, nCount:= 3);
hrSize := fbRepeatedField.CalculateSize(nSize=> nSize);

AssertEquals_DINT(
    Expected:= S_OK,
    Actual:= hr,
    Message:= 'Expected repeated message write to succeed');

AssertArrayEquals_BYTE(
    Expecteds:= cExpected,
    Actuals:= aActual,
    Message:= 'Expected non-packed repeated message wire format');

AssertEquals_DINT(
    Expected:= S_OK,
    Actual:= hrSize,
    Message:= 'Expected repeated message size calculation to succeed');

AssertEquals_UDINT(
    Expected:= 21,
    Actual:= nSize,
    Message:= 'Expected non-packed repeated message size to include tags and message lengths');

TEST_FINISHED_NAMED(__POUNAME());
END_METHOD

END_FUNCTION_BLOCK
